FUNCTION_BLOCK Heating_Ctx_Priv
VAR_INPUT
	iActiveRoom		: I_Room;
END_VAR
VAR_OUTPUT
	iOnEnable		: I_SignalEmit;
	
	iQueue			: I_MutArgQueue;
END_VAR

END_FUNCTION_BLOCK

(* stored: Version 1.1.0.1
   POU Heating_Ctx_Priv: Id {a4dbf3bc-91dd-4988-bf90-c6d789fe1a17}, SpecialFunc None *)
